// TIA Portal project "Proyecto Ascensor" (V17)
// Vorlageprojekt für das Buch mit Zielsystem S7-1200

(* hardware
DEVICE "S7-1200-Station_1"  S7-1200 Station
   slot 0: "Baugruppenträger_0"  Rack  V1.0
   slot 1: "PLC_1"  CPU 1211C DC/DC/DC  6ES7 211-1AE40-0XB0  V4.1
*)

// ===== PLC "PLC_1"  CPU 1211C DC/DC/DC =====

VAR_GLOBAL   // PLC tag table "Standard-Variablentabelle"
   "pulsadorPisoUno" AT %I0.0 : Bool;   // Pulsador del primer piso
   "pulsadorPisoDos" AT %I0.1 : Bool;   // Pulsador del segundo piso
   "pulsadorPisoTres" AT %I0.2 : Bool;   // Pulsador del tercer piso
   "ascensorSube" AT %M5.0 : Bool;   // Marca ascensor subiendo
   "ascensorBaja" AT %M5.1 : Bool;   // Marca ascensor bajando
   "pisoUno" AT %M5.2 : Bool;   // Marca del primer piso
   "pisoDos" AT %M5.3 : Bool;   // Marca del segundo piso
   "pisoTres" AT %M5.4 : Bool;   // Marca del tercer piso
   "sensorUno" AT %I1.0 : Bool;   // Sensor primer piso
   "sensorDos" AT %I1.1 : Bool;   // Sensor segundo piso
   "sensorTres" AT %I1.2 : Bool;   // Sensor tercer piso
   "ledPisoUno" AT %Q0.0 : Bool;   // Luz piloto piso uno
   "ledPisoDos" AT %Q0.1 : Bool;   // Luz piloto piso dos
   "ledPisoTres" AT %Q0.2 : Bool;   // Luz piloto piso tres
   "motorSube" AT %Q0.3 : Bool;   // Motor subiendo
   "motorBaja" AT %Q0.4 : Bool;   // Motor bajando
END_VAR

FUNCTION "MHJ-PLC-Lab-Function-S71200" : Void   // FC9000, SCL
{ S7_Optimized_Access := 'TRUE' }
VERSION : 0.1
   VAR_TEMP
      rdTimeReturn : Int;
      outputTime : DTL;
      SyncVal : Byte;
      forVal : Int;
      forVal_2 : Int;
      Value : Byte;
   END_VAR
   VAR CONSTANT
      CompVal : Byte := 16#34;
      Value_01 : Byte := 16#11;
      Value_01_DW : DWord := 16#A165_D992;
      Value_02_DW : DWord := 16#58BE_4401;
   END_VAR
BEGIN

   #Value:=PEEK(area := 16#82,
        dbNumber := 0,
        byteOffset := 511);
   #Value := #Value + 1;

   POKE(area := 16#82,
        dbNumber := 0,
        byteOffset := 511,
        value := #Value);

   POKE(area:=16#81,
        dbNumber:=0,
        byteOffset:=1016,
        value:=#Value_01_DW);
   POKE(area := 16#81,
        dbNumber := 0,
        byteOffset := 1020,
        value := #Value_02_DW);

   POKE(area := 16#81,
        dbNumber := 0,
        byteOffset := 511,
        value := B#16#00);

   FOR #forVal := 0 TO 120 DO
       FOR #forVal_2:=0 TO 10 DO
           #rdTimeReturn:=RD_SYS_T(#outputTime);
           #rdTimeReturn := WR_SYS_T(#outputTime);
           #rdTimeReturn := RD_SYS_T(#outputTime);
           #rdTimeReturn := WR_SYS_T(#outputTime);
       END_FOR;
       #SyncVal:= PEEK(area := 16#81,
                      dbNumber := 0,
                      byteOffset := 511);
       IF #SyncVal = #CompVal THEN
          GOTO M_1;
       END_IF;
   END_FOR;
   RETURN;

   M_1:
   POKE(area := 16#81,
        dbNumber := 0,
        byteOffset := 511,
        value := B#16#0);
END_FUNCTION

ORGANIZATION_BLOCK "Main"   // OB1, LAD, ProgramCycle
TITLE = "Main Program Sweep (Cycle)"
{ S7_Optimized_Access := 'TRUE' }
VERSION : 0.1
   VAR_INPUT
      Initial_Call : Bool;   // Initial call of this OB
      Remanence : Bool;   // =True, if remanent data are available
   END_VAR
BEGIN

REGION Network 1: Konnektierungsbaustein für PLC-Lab
   // Im Netzwerk 1 wird der Konnektierungsbaustein für PLC-Lab aufgerufen.
   // Dieser Aufruf darf nicht entfernt werden!
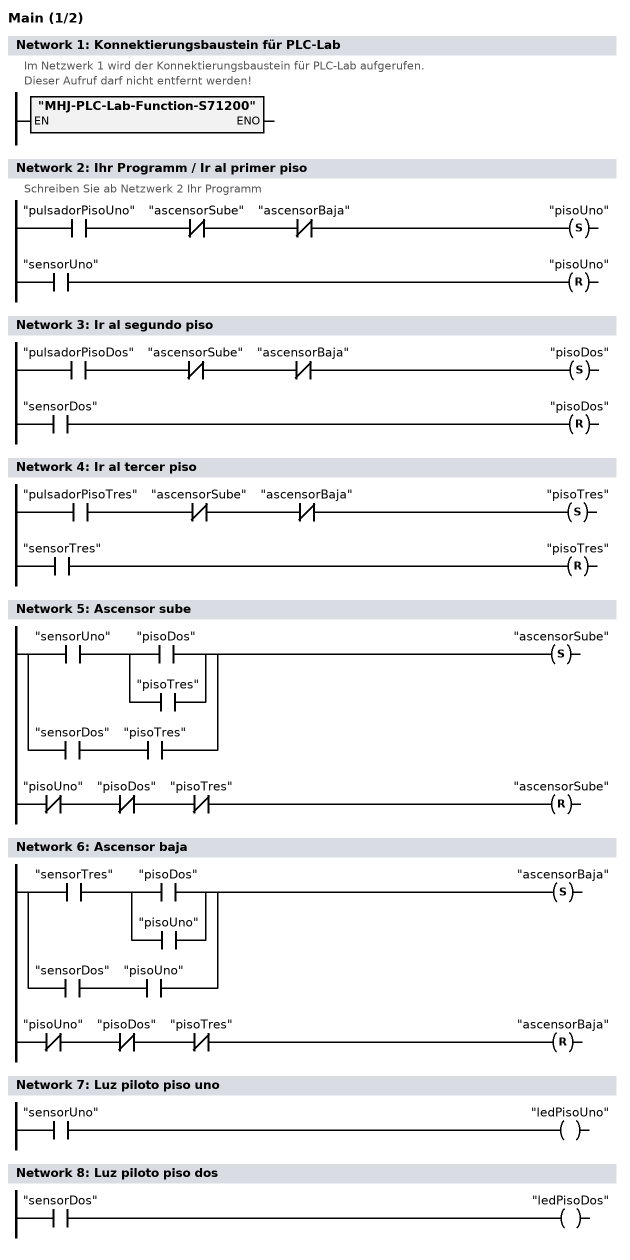
   RUNG wire#powerrail
      "MHJ-PLC-Lab-Function-S71200"()
   END_RUNG
   // the same network as SCL:
   "MHJ-PLC-Lab-Function-S71200"();
END_REGION

REGION Network 2: Ihr Programm / Ir al primer piso
   // Schreiben Sie ab Netzwerk 2 Ihr Programm
   RUNG wire#powerrail
      Contact( "pulsadorPisoUno" )
      I_Contact( "ascensorSube" )
      I_Contact( "ascensorBaja" )
      S_Coil( "pisoUno" )
   END_RUNG
   RUNG wire#powerrail
      Contact( "sensorUno" )
      R_Coil( "pisoUno" )
   END_RUNG
   // the same network as SCL:
   IF "pulsadorPisoUno" AND NOT "ascensorSube" AND NOT "ascensorBaja" THEN "pisoUno" := TRUE; END_IF;
   IF "sensorUno" THEN "pisoUno" := FALSE; END_IF;
END_REGION

REGION Network 3: Ir al segundo piso
   RUNG wire#powerrail
      Contact( "pulsadorPisoDos" )
      I_Contact( "ascensorSube" )
      I_Contact( "ascensorBaja" )
      S_Coil( "pisoDos" )
   END_RUNG
   RUNG wire#powerrail
      Contact( "sensorDos" )
      R_Coil( "pisoDos" )
   END_RUNG
   // the same network as SCL:
   IF "pulsadorPisoDos" AND NOT "ascensorSube" AND NOT "ascensorBaja" THEN "pisoDos" := TRUE; END_IF;
   IF "sensorDos" THEN "pisoDos" := FALSE; END_IF;
END_REGION

REGION Network 4: Ir al tercer piso
   RUNG wire#powerrail
      Contact( "pulsadorPisoTres" )
      I_Contact( "ascensorSube" )
      I_Contact( "ascensorBaja" )
      S_Coil( "pisoTres" )
   END_RUNG
   RUNG wire#powerrail
      Contact( "sensorTres" )
      R_Coil( "pisoTres" )
   END_RUNG
   // the same network as SCL:
   IF "pulsadorPisoTres" AND NOT "ascensorSube" AND NOT "ascensorBaja" THEN "pisoTres" := TRUE; END_IF;
   IF "sensorTres" THEN "pisoTres" := FALSE; END_IF;
END_REGION

REGION Network 5: Ascensor sube
   RUNG wire#powerrail
      Contact( "sensorUno" )
      wire#w1
      Contact( "pisoDos" )
      wire#w2
      S_Coil( "ascensorSube" )
   END_RUNG
   RUNG wire#w1
      Contact( "pisoTres" )
   END_RUNG wire#w2
   RUNG wire#powerrail
      Contact( "sensorDos" )
      Contact( "pisoTres" )
   END_RUNG wire#w2
   RUNG wire#powerrail
      I_Contact( "pisoUno" )
      I_Contact( "pisoDos" )
      I_Contact( "pisoTres" )
      R_Coil( "ascensorSube" )
   END_RUNG
   // the same network as SCL:
   IF ("sensorUno" AND ("pisoDos" OR "pisoTres")) OR ("sensorDos" AND "pisoTres") THEN
       "ascensorSube" := TRUE;
   END_IF;
   IF NOT "pisoUno" AND NOT "pisoDos" AND NOT "pisoTres" THEN "ascensorSube" := FALSE; END_IF;
END_REGION

REGION Network 6: Ascensor baja
   RUNG wire#powerrail
      Contact( "sensorTres" )
      wire#w1
      Contact( "pisoDos" )
      wire#w2
      S_Coil( "ascensorBaja" )
   END_RUNG
   RUNG wire#w1
      Contact( "pisoUno" )
   END_RUNG wire#w2
   RUNG wire#powerrail
      Contact( "sensorDos" )
      Contact( "pisoUno" )
   END_RUNG wire#w2
   RUNG wire#powerrail
      I_Contact( "pisoUno" )
      I_Contact( "pisoDos" )
      I_Contact( "pisoTres" )
      R_Coil( "ascensorBaja" )
   END_RUNG
   // the same network as SCL:
   IF ("sensorTres" AND ("pisoDos" OR "pisoUno")) OR ("sensorDos" AND "pisoUno") THEN
       "ascensorBaja" := TRUE;
   END_IF;
   IF NOT "pisoUno" AND NOT "pisoDos" AND NOT "pisoTres" THEN "ascensorBaja" := FALSE; END_IF;
END_REGION

REGION Network 7: Luz piloto piso uno
   RUNG wire#powerrail
      Contact( "sensorUno" )
      Coil( "ledPisoUno" )
   END_RUNG
   // the same network as SCL:
   "ledPisoUno" := "sensorUno";
END_REGION

REGION Network 8: Luz piloto piso dos
   RUNG wire#powerrail
      Contact( "sensorDos" )
      Coil( "ledPisoDos" )
   END_RUNG
   // the same network as SCL:
   "ledPisoDos" := "sensorDos";
END_REGION

REGION Network 9: Luz piloto piso tres
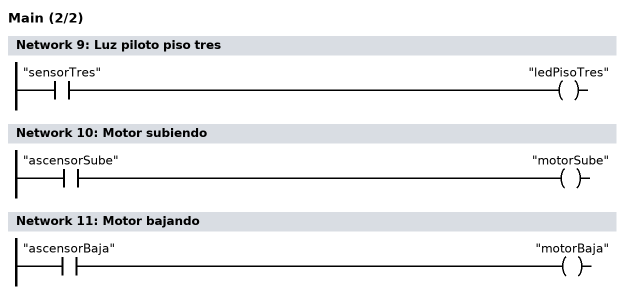
   RUNG wire#powerrail
      Contact( "sensorTres" )
      Coil( "ledPisoTres" )
   END_RUNG
   // the same network as SCL:
   "ledPisoTres" := "sensorTres";
END_REGION

REGION Network 10: Motor subiendo
   RUNG wire#powerrail
      Contact( "ascensorSube" )
      Coil( "motorSube" )
   END_RUNG
   // the same network as SCL:
   "motorSube" := "ascensorSube";
END_REGION

REGION Network 11: Motor bajando
   RUNG wire#powerrail
      Contact( "ascensorBaja" )
      Coil( "motorBaja" )
   END_RUNG
   // the same network as SCL:
   "motorBaja" := "ascensorBaja";
END_REGION
END_ORGANIZATION_BLOCK